{attribute 'global_init_slot' := '40510'}
VAR_GLOBAL
  LblControl_OperationMode                                     :FB_BA_Label:=( sObjName:='OPM',sDescr:='Operation Mode');
  LblControl_SummerNightCooling                                :FB_BA_Label:=( sObjName:='SNC',sDescr:='Summer night cooling');
  LblControl_DifferencePressureMonitoringSupplyAirFan          :FB_BA_Label:=( sObjName:='DPM',sDescr:='Difference Pressure Monitoring Supply Air Fan');
  LblControl_DifferencePressureMonitoringExtractAirFan         :FB_BA_Label:=( sObjName:='DPM',sDescr:='Difference Pressure Monitoring Extract Air Fan');
  LblControl_TSetpointCalculation                              :FB_BA_Label:=( sObjName:='SPC',sDescr:='Setpoint Calculation Temperature');
  LblControl_HSetpointCalculation                              :FB_BA_Label:=( sObjName:='SPC',sDescr:='Setpoint Calculation Humidity');
  LblControl_TCascadeSupplyAirControl                          :FB_BA_Label:=( sObjName:='CTL',sDescr:='Cascade control supply air temperature');
  LblControl_HCascadeSupplyAirControl                          :FB_BA_Label:=( sObjName:='CTL',sDescr:='Cascade control supply air humidity');
  LblControl_PreHeater                                         :FB_BA_Label:=( sObjName:='PRH',sDescr:='PreHeater');
  LblControl_ReHeater                                          :FB_BA_Label:=( sObjName:='RHE',sDescr:='Reheater');
  LblControl_EnergyRecovery                                    :FB_BA_Label:=( sObjName:='ERC',sDescr:='Energy Recovery');
  LblControl_SupplyAirTemperatureControl                       :FB_BA_Label:=( sObjName:='CTL',sDescr:='Supply Air Temperature Control');
  LblControl_SupplyAirDehumidifierControl                      :FB_BA_Label:=( sObjName:='CTL',sDescr:='Supply Air Dehumidification Control');
  LblControl_SupplyAirHumidifierController                     :FB_BA_Label:=( sObjName:='CTL',sDescr:='Supply Air Humidity Control');
  LblControl_SupplyAirTemperatureLimitationControl             :FB_BA_Label:=( sObjName:='CTL',sDescr:='Supply Air Temperature Limitation Control');
  LblControl_ReturnWaterControl                                :FB_BA_Label:=( sObjName:='CTL',sDescr:='Return Water Control');
  LblControl_HumidityLimitationControl                         :FB_BA_Label:=( sObjName:='CTL',sDescr:='Rel humidity limitation control');
  LblControl_CalculationPreRinseSetpoint                       :FB_BA_Label:=( sObjName:='SPC',sDescr:='Calculation PreRinse Setpoint');
  LblControl_FrostProtectionControl                            :FB_BA_Label:=( sObjName:='FPC',sDescr:='Frost Protection Control');
  LblControl_ExhaustAirTemperatureControl                      :FB_BA_Label:=( sObjName:='CTL',sDescr:='Exhaust Air Temperature Control');
  LblControl_EnergyRecoveryDeicingRamp                         :FB_BA_Label:=( sObjName:='RMP',sDescr:='Energy Recovery Deicing Ramp');
  LblControl_BACnetDevice                                      :FB_BA_Label:=( sObjName:='DEV',sDescr:='BACnet device');
  LblControl_PlantControl                                      :FB_BA_Label:=( sObjName:='PCT',sDescr:='Plant Control');
  LblControl_TSequenceControl                                  :FB_BA_Label:=( sObjName:='SEQ',sDescr:='Sequence Control Temp');
  LblControl_HSequenceControl                                  :FB_BA_Label:=( sObjName:='SEQ',sDescr:='Sequence Control Humidity');
  LblControl_GeneralBeckhoffEventClass                         :FB_BA_Label:=( sObjName:='ECL',sDescr:='Event class');
  LblControl_GeneralSettings                                   :FB_BA_Label:=( sObjName:='SYP',sDescr:='System parameters');
  LblControl_GeneralCabinetBasicEquipment                      :FB_BA_Label:=( sObjName:='CBE',sDescr:='Cabinet basic equipment');
  LblControl_GeneralCabinetAdditionalEquipment                 :FB_BA_Label:=( sObjName:='CAE',sDescr:='Cabinet additional equipment');
  LblControl_EventIndicationLamp                               :FB_BA_Label:=( sObjName:='CEM',sDescr:='Collective error message lamp');
  LblControl_AcknowledgeCommand                                :FB_BA_Label:=( sObjName:='ACK',sDescr:='Acknowledge Hardware');
  LblControl_RemoteAcknowledgement                             :FB_BA_Label:=( sObjName:='ACK',sDescr:='Remote acknowledgement fault');
  LblControl_LocalAcknowledgement                              :FB_BA_Label:=( sObjName:='ACK',sDescr:='Local acknowledgement fault');
  LblControl_Acknowledge                                       :FB_BA_Label:=( sObjName:='ACK',sDescr:='Acknowledge');
// 
  LblControl_Fuse                                              :FB_BA_Label:=( sObjName:='FUS',sDescr:='Fuse');
// Settings
  LblControl_FrostProtection                                   :FB_BA_Label:=( sObjName:='FRP',sDescr:='Frost protection');
  LblControl_MinimumOutsideTemperature                         :FB_BA_Label:=( sObjName:='TWT',sDescr:='Minimum outdoor temperature');
  LblControl_TemperatureWeatherLowLimit                        :FB_BA_Label:=( sObjName:='TWT',sDescr:='Temperature weather low limit');
  LblControl_TemperatureWeatherDamped                          :FB_BA_Label:=( sObjName:='TWD',sDescr:='Temperature weather damped');
  LblControl_TemperatureWeatherDampedLowLimit                  :FB_BA_Label:=( sObjName:='TWD',sDescr:='Temperature Weather damped low limit');
  LblControl_PressureControl                                   :FB_BA_Label:=( sObjName:='CTL',sDescr:='Pressure control');
  LblControl_Converter3Point                                   :FB_BA_Label:=( sObjName:='CNV',sDescr:='3 point converter');
  LblControl_HeatingCurve                                      :FB_BA_Label:=( sObjName:='HCV',sDescr:='Heating curve');
  LblControl_SetpointGeneration                                :FB_BA_Label:=( sObjName:='SPG',sDescr:='Setpoint generation');
  LblControl_RequestHeatState                                  :FB_BA_Label:=( sObjName:='RHS',sDescr:='Request heat state');
  LblControl_RequestHeatSetpoint                               :FB_BA_Label:=( sObjName:='RHS',sDescr:='Request heat setpoint');
  LblControl_FlowTempControl                                   :FB_BA_Label:=( sObjName:='CTL',sDescr:='Flow temperature control');
// 
  LblControl_RoomTemperatureControl                            :FB_BA_Label:=( sObjName:='RGL',sDescr:='Room Temperature Control');
  LblControl_FlowTemperatureControl                            :FB_BA_Label:=( sObjName:='CTL',sDescr:='Flow temperature control');
  LblControl_SetpointHeating                                   :FB_BA_Label:=( sObjName:='SPG',sDescr:='Setpoint generation heating');
  LblControl_SetpointCooling                                   :FB_BA_Label:=( sObjName:='SPG',sDescr:='Setpoint generation cooling');
  LblControl_Facade                                            :FB_BA_Label:=( sObjName:='FIE',sDescr:='Facade Data');
  LblControl_BuildingAlarms                                    :FB_BA_Label:=( sObjName:='FIE',sDescr:='Building Alarms');
  LblControl_BuildingEnergyLevel                               :FB_BA_Label:=( sObjName:='FIE',sDescr:='Building Energylevel');
  LblControl_BuildingMode                                      :FB_BA_Label:=( sObjName:='FIE',sDescr:='Building Operationmode');
  LblControl_BuildingSpRmT                                     :FB_BA_Label:=( sObjName:='FIE',sDescr:='Building Roomtemperature Setpoints');
  LblControl_BuildingSunprotection                             :FB_BA_Label:=( sObjName:='FIE',sDescr:='Building Sunprotection');
  LblControl_TemperatureFrost                                  :FB_BA_Label:=( sObjName:='TFR',sDescr:='Temperature Frost');
  LblControl_MixedAirStartUpRamp                               :FB_BA_Label:=( sObjName:='RMP',sDescr:='Ramp plant start');
  LblControl_Cooler                                            :FB_BA_Label:=( sObjName:='COL',sDescr:='Cooler');
  LblControl_EvtCategoryLifeSafty                              :FB_BA_Label:=( sObjName:='EDL',sDescr:='Danger to life');
  LblControl_EvtCategorySaftyMessage                           :FB_BA_Label:=( sObjName:='ESM',sDescr:='Safety message');
  LblControl_EvtCategoryAlarmMessage                           :FB_BA_Label:=( sObjName:='EAM',sDescr:='Alarm message');
  LblControl_EvtCategoryFaultMessage                           :FB_BA_Label:=( sObjName:='EFM',sDescr:='Fault message');
  LblControl_EvtCategoryMaintenanceMessage                     :FB_BA_Label:=( sObjName:='EMM',sDescr:='Maintenance message');
  LblControl_EvtCategorySystem                                 :FB_BA_Label:=( sObjName:='ESY',sDescr:='System message');
  LblControl_EvtCategoryManualOperation                        :FB_BA_Label:=( sObjName:='EMO',sDescr:='Manual operation');
  LblControl_EvtCategoryOther                                  :FB_BA_Label:=( sObjName:='EOM',sDescr:='Other message');
  LblControl_TrendLogging                                      :FB_BA_Label:=( sObjName:='TRL',sDescr:='TrendLogging                                      ');
  LblControl_WeatherParameters                                 :FB_BA_Label:=( sObjName:='WTP',sDescr:='Weather Parameters');
  LblControl_SetpointFrostProtection                           :FB_BA_Label:=( sObjName:='SP_',sDescr:='Setpoint frost protection');
  LblControl_SetpointWeatherIcing                              :FB_BA_Label:=( sObjName:='SP_',sDescr:='Setpoint icing');
  LblControl_SetpointMinimumOutsideTemperature                 :FB_BA_Label:=( sObjName:='SPI',sDescr:='Setpoint minimum outside temperature');
  LblControl_MeanDamped                                        :FB_BA_Label:=( sObjName:='MWD',sDescr:='Mean value weather temperature damped');
  LblControl_OperationalMessageTemperatureWeatherLowLimit      :FB_BA_Label:=( sObjName:='OM_',sDescr:='Operational Message Temperature Weather Low Limit');
  LblControl_OperationalMessageTemperatureWeatherDampedLowLimit:FB_BA_Label:=( sObjName:='OM_',sDescr:='Operational Message Temperature Weather Damped Low Limit');
// Beckhoff Cabinet basic equipment
  LblControl_SwitchingCommandCollectiveFaultSignalLamp         :FB_BA_Label:=( sObjName:='SC_',sDescr:='Collective fault signal lamp switching command');
  LblControl_SwitchingCommandHardwareAcknowledgement           :FB_BA_Label:=( sObjName:='SC_',sDescr:='Hardware acknowledgement switching command');
  LblControl_ButtonRemoteAcknowledgement                       :FB_BA_Label:=( sObjName:='BUT',sDescr:='Input remote acknowledgement');
  LblControl_ButtonLocalAcknowledgement                        :FB_BA_Label:=( sObjName:='BUT',sDescr:='Button acknowledgement');
// Beckhoff Heating Circuit
  LblControl_HeatingLimit                                      :FB_BA_Label:=( sObjName:='HLM',sDescr:='Heating limit ');
  LblControl_PresentOperationMode                              :FB_BA_Label:=( sObjName:='POM',sDescr:='Present operation mode');
  LblControl_OperationModeSelection                            :FB_BA_Label:=( sObjName:='OMS',sDescr:='Operation mode selection');
// Beckhoff Summer Night Cooling
  LblControl_HysteresisRoomTemperature                         :FB_BA_Label:=( sObjName:='HYS',sDescr:='Hyeresis room temperature');
  LblControl_OutsideTemperatureLowLimit                        :FB_BA_Label:=( sObjName:='MIN',sDescr:='minimum outside temperature');
  LblControl_OffValueDifferenceOutsideInsightTemperature       :FB_BA_Label:=( sObjName:='MIN',sDescr:='Off Value differenz between ouside and insight temperature');
  LblControl_OnValueDifferenceOutsideInsightTemperature        :FB_BA_Label:=( sObjName:='MAX',sDescr:='On Value differenz between ouside and insight temperature');
// Beckhoff Damper
  LblControl_DriveTimeOpen                                     :FB_BA_Label:=( sObjName:='DTO',sDescr:='Drive time open');
  LblControl_DriveTimeClose                                    :FB_BA_Label:=( sObjName:='DTC',sDescr:='Drive time close');
  LblControl_DisturbanceFeedbackOpen                           :FB_BA_Label:=( sObjName:='DSO',sDescr:='Disturbance_feedback_open');
  LblControl_DisturbanceFeedbackClose                          :FB_BA_Label:=( sObjName:='DSC',sDescr:='Disturbance_feedback_close');
// 
  LblControl_TimeDelay                                         :FB_BA_Label:=( sObjName:='TD_',sDescr:='Time delay ');
  LblControl_TimeDelayFeedback                                 :FB_BA_Label:=( sObjName:='TDF',sDescr:='Time delay feedback');
  LblControl_TimeDelayInterruptionFeedback                     :FB_BA_Label:=( sObjName:='TDI',sDescr:='Time delay interruption');
// Beckhoff pre rins
  LblControl_PreRinseDuration                                  :FB_BA_Label:=( sObjName:='PRD',sDescr:='Pre rins duration');
  LblControl_DisturbancePreRinse                               :FB_BA_Label:=( sObjName:='DST',sDescr:='Disturbance pre rinse');
  LblControl_SetpointMinimalReturnWaterTemperature             :FB_BA_Label:=( sObjName:='SP_',sDescr:='Setpoint minimal return water temperature');
// Beckhoff ramp 
  LblControl_RampTimeUp                                        :FB_BA_Label:=( sObjName:='RTU',sDescr:='Ramp time up');
  LblControl_RampTimeDown                                      :FB_BA_Label:=( sObjName:='RTD',sDescr:='Ramp time down');
  LblControl_CommandOpen                                       :FB_BA_Label:=( sObjName:='SC_',sDescr:='Switch command open');
  LblControl_CommandClose                                      :FB_BA_Label:=( sObjName:='SC_',sDescr:='Switch command close');
  LblControl_CalculatedValue                                   :FB_BA_Label:=( sObjName:='CAV',sDescr:='calculated value');
  LblControl_Value                                             :FB_BA_Label:=( sObjName:='VAL',sDescr:='Value');
// Beckhoff event class
  LblControl_EvtClass                                          :FB_BA_Label:=( sObjName:='NC_',sDescr:='Notification class');
  LblControl_FlowSwitch                                        :FB_BA_Label:=( sObjName:='OM_',sDescr:='Operating message flow monitor');
  LblControl_SmokeAlarm                                        :FB_BA_Label:=( sObjName:='DST',sDescr:='Disturbance smoke alarm');
  LblControl_SystemFailure                                     :FB_BA_Label:=( sObjName:='DST',sDescr:='Disturbance system failure');
  LblControl_Contamination                                     :FB_BA_Label:=( sObjName:='DST',sDescr:='Disturbance Contamination');
  LblControl_SwitchingCommandSmokeDetector                     :FB_BA_Label:=( sObjName:='SC_',sDescr:='Switching command acknowledge');
  LblControl_ButtonReset                                       :FB_BA_Label:=( sObjName:='BUT',sDescr:='Button acknowledge');
  LblControl_OffsetNightSetpoint                               :FB_BA_Label:=( sObjName:='ONS',sDescr:='Offset night setback');
// 
  LblControl_SetpointRelHumidityHumidification                 :FB_BA_Label:=( sObjName:='SP_',sDescr:='Setpoint Relative Humidity Humidification');
  LblControl_SetpointRelHumidityDehumidification               :FB_BA_Label:=( sObjName:='SP_',sDescr:='Setpoint Relative Humidity Dehumidification');
  LblControl_SetpointAbsHumidityHumidification                 :FB_BA_Label:=( sObjName:='SPC',sDescr:='Setpoint absolute humidity humidification');
  LblControl_SetpointAbsHumidityDehumidification               :FB_BA_Label:=( sObjName:='SPC',sDescr:='Setpoint absolute humidity dehumidification');
  LblControl_SetpointRelHumidity                               :FB_BA_Label:=( sObjName:='SP_',sDescr:='Setpoint relative humidity');
  LblControl_SetpointAbsHumidity                               :FB_BA_Label:=( sObjName:='SP_',sDescr:='Setpoint absolute humidity');
  LblControl_OperationalMessageDehumidification                :FB_BA_Label:=( sObjName:='OM_',sDescr:='Operational message dehumidification');
// 
  LblControl_SetpointSunblindPosition                          :FB_BA_Label:=( sObjName:='SP_',sDescr:='Setpoint blind position');
  LblControl_SetpointSunblindAngle                             :FB_BA_Label:=( sObjName:='SP_',sDescr:='Setpoint blind angle');
  LblControl_CommandSunblindStart                              :FB_BA_Label:=( sObjName:='SC_',sDescr:='Command sunblind start');
  LblControl_ButtonSunblind                                    :FB_BA_Label:=( sObjName:='BUT',sDescr:='Sun blind button');
  LblControl_FeedbackSunblindPosition                          :FB_BA_Label:=( sObjName:='FDB',sDescr:='Feedback blind position');
  LblControl_FeedbackSunblindAngle                             :FB_BA_Label:=( sObjName:='FDB',sDescr:='Feedback blind angle');
  LblControl_FeedbackSunblindPrio                              :FB_BA_Label:=( sObjName:='FDB',sDescr:='Feedback Telegram-Priority');
// 
  LblControl_TimeDelayStormOn                                  :FB_BA_Label:=( sObjName:='TON',sDescr:='Storm-detection time delay on');
  LblControl_TimeDelayStormOff                                 :FB_BA_Label:=( sObjName:='TOF',sDescr:='Storm-detection time delay off');
  LblControl_MaintenanceEnable                                 :FB_BA_Label:=( sObjName:='EN_',sDescr:='Maintenence positioning enable');
  LblControl_MaintenancePosition                               :FB_BA_Label:=( sObjName:='SP_',sDescr:='Setpoint maintenance position');
  LblControl_MaintenanceAngle                                  :FB_BA_Label:=( sObjName:='SP_',sDescr:='Setpoint maintenance angle');
  LblControl_FacadeThermoAutomaticEnable                       :FB_BA_Label:=( sObjName:='EN_',sDescr:='Facade-Thermoautomatic enable');
  LblControl_FacadeThermoAutomaticCoolingPosition              :FB_BA_Label:=( sObjName:='SP_',sDescr:='Facade-Thermoautomatic cooling-position');
  LblControl_FacadeThermoAutomaticCoolingAngle                 :FB_BA_Label:=( sObjName:='SP_',sDescr:='Facade-Thermoautomatic cooling-angle');
  LblControl_FacadeTwilightAutomaticEnable                     :FB_BA_Label:=( sObjName:='EN_',sDescr:='Facade-Twilightautomatic enable');
  LblControl_SunProtectionValueOn                              :FB_BA_Label:=( sObjName:='SP_',sDescr:='Sun-protection brightness on');
  LblControl_SunProtectionValueOff                             :FB_BA_Label:=( sObjName:='SP_',sDescr:='Sun-protection brightness off');
  LblControl_TimeDelaySunProtectionOn                          :FB_BA_Label:=( sObjName:='TON',sDescr:='Sun-protection brightness on');
  LblControl_TimeDelaySunProtectionOff                         :FB_BA_Label:=( sObjName:='TOF',sDescr:='Sun-protection brightness off');
  LblControl_FacadeParkingEnable                               :FB_BA_Label:=( sObjName:='EN_',sDescr:='Facade-parking enable');
  LblControl_FacadeParkingPosition                             :FB_BA_Label:=( sObjName:='SP_',sDescr:='Facade-parking position');
  LblControl_FacadeParkingAngle                                :FB_BA_Label:=( sObjName:='SP_',sDescr:='Facade-parking angle');
  LblControl_WindProtectionState                               :FB_BA_Label:=( sObjName:='STA',sDescr:='State wind-protection');
  LblControl_SunProtectionState                                :FB_BA_Label:=( sObjName:='STA',sDescr:='State sun-protection');
// 
  LblControl_LowWaterMonitor                                   :FB_BA_Label:=( sObjName:='DST',sDescr:='Low water monitor');
  LblControl_FireAlert                                         :FB_BA_Label:=( sObjName:='DST',sDescr:='Fire alert');
  LblControl_Burglary                                          :FB_BA_Label:=( sObjName:='DST',sDescr:='Burglary alert');
  LblControl_CentralSwitchOff                                  :FB_BA_Label:=( sObjName:='PLS',sDescr:='Central switch-off');
  LblControl_ForcedVentilation                                 :FB_BA_Label:=( sObjName:='PLS',sDescr:='Forced ventilation ');
  LblControl_SmokeExtraction                                   :FB_BA_Label:=( sObjName:='PLS',sDescr:='Smoke extraction');
  LblControl_SetpointIce                                       :FB_BA_Label:=( sObjName:='SP_',sDescr:='Setpoint Ice');
  LblControl_SunProtectionInterval                             :FB_BA_Label:=( sObjName:='SP_',sDescr:='Sun-protection positioning interval');
  LblControl_DeiceTime                                         :FB_BA_Label:=( sObjName:='SP_',sDescr:='Frost-protection deice-time');
  LblControl_GlobalThermoAutomaticValueOn                      :FB_BA_Label:=( sObjName:='SP_',sDescr:='Thermo-automatic radiation-value on');
  LblControl_GlobalThermoAutomaticValueOff                     :FB_BA_Label:=( sObjName:='SP_',sDescr:='Thermo-automatic radiation-value off');
  LblControl_GlobalTwilightAutomaticValueOn                    :FB_BA_Label:=( sObjName:='SP_',sDescr:='Twilight-automatic brightness-value on');
  LblControl_GlobalTwilightAutomaticValueOff                   :FB_BA_Label:=( sObjName:='SP_',sDescr:='Twilight-automatic brightness-value on');
  LblControl_IceAlert                                          :FB_BA_Label:=( sObjName:='DST',sDescr:='Ice alert');
  LblControl_GlobalThermoAutomaticRelease                      :FB_BA_Label:=( sObjName:='EN_',sDescr:='Thermo-automatic release');
  LblControl_GlobalTwilightAutomaticRelease                    :FB_BA_Label:=( sObjName:='EN_',sDescr:='Twilight-automatic release');
  LblControl_GlobalResetManMode                                :FB_BA_Label:=( sObjName:='PLS',sDescr:='Global Reset Manual Mode');
// 
  LblControl_BuildingEnergyLevelManual                         :FB_BA_Label:=( sObjName:='OPS',sDescr:='Building-energy-level manual selection');
  LblControl_BuildingEnergyLevelActual                         :FB_BA_Label:=( sObjName:='POM',sDescr:='Building-energy-level actual selection');
  LblControl_BuildingEnergyLevelSched                          :FB_BA_Label:=( sObjName:='SCH',sDescr:='Building-energy-level scheduler');
  LblControl_BuildingModeManual                                :FB_BA_Label:=( sObjName:='OPS',sDescr:='Building-mode manual selection');
  LblControl_BuildingModeActual                                :FB_BA_Label:=( sObjName:='POM',sDescr:='Building-mode actual selection');
  LblControl_BuildingModeSched                                 :FB_BA_Label:=( sObjName:='SCH',sDescr:='Building-mode scheduler');
// 
  LblControl_SummerCompensationX1                              :FB_BA_Label:=( sObjName:='IPX',sDescr:='Summercompensation X1');
  LblControl_SummerCompensationX2                              :FB_BA_Label:=( sObjName:='IPX',sDescr:='Summercompensation X2');
  LblControl_SummerCompensationY1                              :FB_BA_Label:=( sObjName:='IPY',sDescr:='Summercompensation Y1');
  LblControl_SummerCompensationY2                              :FB_BA_Label:=( sObjName:='IPY',sDescr:='Summercompensation Y2');
  LblControl_WinterCompensationX1                              :FB_BA_Label:=( sObjName:='IPX',sDescr:='Wintercompensation X1');
  LblControl_WinterCompensationX2                              :FB_BA_Label:=( sObjName:='IPX',sDescr:='Wintercompensation X2');
  LblControl_WinterCompensationY1                              :FB_BA_Label:=( sObjName:='IPY',sDescr:='Wintercompensation Y1');
  LblControl_WinterCompensationY2                              :FB_BA_Label:=( sObjName:='IPY',sDescr:='Wintercompensation Y2');
  LblControl_SummerCompensation                                :FB_BA_Label:=( sObjName:='SCP',sDescr:='SummerCompensation');
  LblControl_WinterCompensation                                :FB_BA_Label:=( sObjName:='WCP',sDescr:='WinterCompensation');
  LblControl_SummerCompensationYmin                            :FB_BA_Label:=( sObjName:='SPI',sDescr:='Summer Compensation Ymin');
  LblControl_SummerCompensationYmax                            :FB_BA_Label:=( sObjName:='SPX',sDescr:='Summer Compensation Ymax');
  LblControl_WinterCompensationYmin                            :FB_BA_Label:=( sObjName:='SPI',sDescr:='Winter Compensation Ymin');
  LblControl_WinterCompensationYmax                            :FB_BA_Label:=( sObjName:='SPX',sDescr:='Winter Compensation Ymax');
  LblControl_SummerCompensationSp                              :FB_BA_Label:=( sObjName:='SPC',sDescr:='Summer Compensation Setpoint');
  LblControl_WinterCompensationSp                              :FB_BA_Label:=( sObjName:='SPC',sDescr:='Winter Compensation Setpoint');
  LblControl_SetpointShiftHeating                              :FB_BA_Label:=( sObjName:='SP_',sDescr:='Setpoint shift heating');
  LblControl_SetpointShiftCooling                              :FB_BA_Label:=( sObjName:='SP_',sDescr:='Setpoint shift cooling');
  LblControl_DampConstant                                      :FB_BA_Label:=( sObjName:='SP_',sDescr:='Damp constant');
// 
  LblControl_DelayOn                                           :FB_BA_Label:=( sObjName:='TON',sDescr:='Switch-on delay');
  LblControl_DelayOff                                          :FB_BA_Label:=( sObjName:='TOF',sDescr:='Switch-off delay');
  LblControl_AntiBlocking                                      :FB_BA_Label:=( sObjName:='ABK',sDescr:='Anti Blocking');
  LblControl_IdlePeriod                                        :FB_BA_Label:=( sObjName:='ITV',sDescr:='Idle Period');
  LblControl_ImpulsLength                                      :FB_BA_Label:=( sObjName:='IPL',sDescr:='Impuls length');
  LblControl_SuppyAirTempSetpointHeaterCalc                    :FB_BA_Label:=( sObjName:='SPC',sDescr:='Suppy Air Sp Heater Calc');
  LblControl_SuppyAirTempSetpointCoolerCalc                    :FB_BA_Label:=( sObjName:='SPC',sDescr:='Suppy Air Sp Cooler Calc');
  LblControl_SuppyAirTempSetpointERCCalc                       :FB_BA_Label:=( sObjName:='SPC',sDescr:='Suppy Air Sp ERC Calc');
  LblControl_X01                                               :FB_BA_Label:=( sObjName:='SPX',sDescr:='Value Base [X1]');
  LblControl_X02                                               :FB_BA_Label:=( sObjName:='SPX',sDescr:='Value Base [X2]');
  LblControl_X03                                               :FB_BA_Label:=( sObjName:='SPX',sDescr:='Value Base [X3]');
  LblControl_X04                                               :FB_BA_Label:=( sObjName:='SPX',sDescr:='Value Base [X4]');
  LblControl_X05                                               :FB_BA_Label:=( sObjName:='SPX',sDescr:='Value Base [X5]');
  LblControl_X06                                               :FB_BA_Label:=( sObjName:='SPX',sDescr:='Value Base [X6]');
  LblControl_X07                                               :FB_BA_Label:=( sObjName:='SPX',sDescr:='Value Base [X7]');
  LblControl_Y01                                               :FB_BA_Label:=( sObjName:='SPY',sDescr:='Value Base [Y1]');
  LblControl_Y02                                               :FB_BA_Label:=( sObjName:='SPY',sDescr:='Value Base [Y2]');
  LblControl_Y02_03                                            :FB_BA_Label:=( sObjName:='SPY',sDescr:='Value Base [Y2Y3]');
  LblControl_Y03                                               :FB_BA_Label:=( sObjName:='SPY',sDescr:='Value Base [Y3]');
  LblControl_Y04                                               :FB_BA_Label:=( sObjName:='SPY',sDescr:='Value Base [Y4]');
  LblControl_Y05                                               :FB_BA_Label:=( sObjName:='SPY',sDescr:='Value Base [Y5]');
  LblControl_Y06                                               :FB_BA_Label:=( sObjName:='SPY',sDescr:='Value Base [Y6]');
  LblControl_Y07                                               :FB_BA_Label:=( sObjName:='SPY',sDescr:='Value Base [Y7]');
  LblControl_FeedbackMonitoring                                :FB_BA_Label:=( sObjName:='FDM',sDescr:='Feedback monitoring');
  LblControl_PreAlarmLimitMAX                                  :FB_BA_Label:=( sObjName:='LMX',sDescr:='Pre Alarm Limit MAX');
  LblControl_PreAlarmLimitMIN                                  :FB_BA_Label:=( sObjName:='LMI',sDescr:='Pre Alarm Limit MIN');
  LblControl_PreAlarmFault                                     :FB_BA_Label:=( sObjName:='DST',sDescr:='Pre Alarm Fault');
  LblControl_MainAlarmLimitMAX                                 :FB_BA_Label:=( sObjName:='LMX',sDescr:='Main Alarm Limit MAX');
  LblControl_MainAlarmLimitMIN                                 :FB_BA_Label:=( sObjName:='LMI',sDescr:='Main Alarm Limit MIN');
  LblControl_MainAlarmFault                                    :FB_BA_Label:=( sObjName:='DST',sDescr:='Main Alarm Fault');
  LblControl_ProcPreRinse                                      :FB_BA_LabelProcess:=( sProcessName:='Process Pre Rinse');
  LblControl_ProjectInfo                                       :FB_BA_Label:=( sObjName:='PI_',sDescr:='Project Info');
END_VAR

// ---- Templates/GVLs/Language/English/LblFunctions_EN.TcGVL
{region '#Template'}
	{attribute 'Version' := '1.2.0.0'}
	{attribute 'Tags' := '"LCID": "1031", "Text": "GVL, AKS, Labels, ObjectName, Description"'}
	{attribute 'Tags' := '"LCID": "1033", "Text": "GVL, DPAD, Labels, ObjectName, Description"'}
	{attribute 'Description' := '"LCID": "1031", "Text": "Anlagenkennzeichnungssystem, Labels functions"'}
	{attribute 'Description' := '"LCID": "1033", "Text": "Data Point Addressing Description, Labels functions"'}
{endregion}

{attribute 'global_init_slot' := '40510'}
VAR_GLOBAL
  LblFunctions_Requirement                                       :FB_BA_Label:=( sObjName:='REQ',sDescr:='Requirement');
  LblFunctions_SystemSwitch                                      :FB_BA_Label:=( sObjName:='PLS',sDescr:='Plant switch');
  LblFunctions_StatusOccupiedRoom                                :FB_BA_Label:=( sObjName:='OCC',sDescr:='Occupied status room');
  LblFunctions_LimitCalculatedValue                              :FB_BA_Label:=( sObjName:='LMC',sDescr:='Calculated limit value');
  LblFunctions_SetpointCalculated                                :FB_BA_Label:=( sObjName:='SPC',sDescr:='Calculated setpoint');
  LblFunctions_ReadyForOperation                                 :FB_BA_Label:=( sObjName:='RFO',sDescr:='Ready for operation');
  LblFunctions_OperationalMessage                                :FB_BA_Label:=( sObjName:='OM_',sDescr:='Operational message');
  LblFunctions_HoursOfOperation                                  :FB_BA_Label:=( sObjName:='OH_',sDescr:='Operating hours');
  LblFunctions_LimitValueHoursOfOperation                        :FB_BA_Label:=( sObjName:='OHL',sDescr:='Operating hours limit value');
  LblFunctions_ObjectCalendar                                    :FB_BA_Label:=( sObjName:='CAL',sDescr:='Calendar object');
  LblFunctions_ObjectCommand                                     :FB_BA_Label:=( sObjName:='COM',sDescr:='Command object');
  LblFunctions_DifferentialConstantController                    :FB_BA_Label:=( sObjName:='TV_',sDescr:='Differential constant controller');
  LblFunctions_SwitchOnErrorUnauthorisedON                       :FB_BA_Label:=( sObjName:='SWE',sDescr:='Switch-on error, unauthorised ON');
  LblFunctions_EnergyLevel                                       :FB_BA_Label:=( sObjName:='EL_',sDescr:='Energy level');
  LblFunctions_EnergyLevelCalculated                             :FB_BA_Label:=( sObjName:='ELC',sDescr:='Energy level calculated');
  LblFunctions_UnlockingDevice                                   :FB_BA_Label:=( sObjName:='UNL',sDescr:='Unlocking device');
  LblFunctions_ObjectEventEnrollment                             :FB_BA_Label:=( sObjName:='EE_',sDescr:='Event enrollment object');
  LblFunctions_Enabled                                           :FB_BA_Label:=( sObjName:='EN_',sDescr:='Enabled');
  LblFunctions_DangerAlarm                                       :FB_BA_Label:=( sObjName:='DA_',sDescr:='Danger alarm');
  LblFunctions_Threshold                                         :FB_BA_Label:=( sObjName:='LM_',sDescr:='Limit value');
  LblFunctions_LimitMAX                                          :FB_BA_Label:=( sObjName:='LMX',sDescr:='MAX limit');
  LblFunctions_LimitMIN                                          :FB_BA_Label:=( sObjName:='LMI',sDescr:='MIN limit');
  LblFunctions_LimitNight                                        :FB_BA_Label:=( sObjName:='LMN',sDescr:='Night limit');
  LblFunctions_LimitDay                                          :FB_BA_Label:=( sObjName:='LMD',sDescr:='Day limit');
  LblFunctions_ObjectGroup                                       :FB_BA_Label:=( sObjName:='GP_',sDescr:='Group object');
  LblFunctions_localPriorityAndOperatingUnitsManualMessage       :FB_BA_Label:=( sObjName:='MNM',sDescr:='local priority and operating units manual message');
  LblFunctions_HeatingCharacteristicCurveExponent                :FB_BA_Label:=( sObjName:='HEX',sDescr:='Heating characteristic curve exponent');
  LblFunctions_HeatingCharacteristicCurveParallelDisplacement    :FB_BA_Label:=( sObjName:='HPD',sDescr:='Heating characteristic curve parallel displacement');
  LblFunctions_HeatingCharacteristicCurveSteepness               :FB_BA_Label:=( sObjName:='HST',sDescr:='Heating characteristic curve steepness');
  LblFunctions_HeatingCircuitNightReduction                      :FB_BA_Label:=( sObjName:='NGT',sDescr:='Heating circuit night reduction');
  LblFunctions_Hysteresis                                        :FB_BA_Label:=( sObjName:='HYS',sDescr:='Hysteresis');
  LblFunctions_Calendar                                          :FB_BA_Label:=( sObjName:='CAL',sDescr:='Calendar');
  LblFunctions_RuntimeError                                      :FB_BA_Label:=( sObjName:='RUN',sDescr:='Runtime error');
  LblFunctions_LoopMAXLimit                                      :FB_BA_Label:=( sObjName:='LPX',sDescr:='Loop MAX limit');
  LblFunctions_LoopMINLimit                                      :FB_BA_Label:=( sObjName:='LPI',sDescr:='Loop MIN limit');
  LblFunctions_LoopObject                                        :FB_BA_Label:=( sObjName:='LP_',sDescr:='Loop object (controller object) – complex object');
  LblFunctions_LoopObjectCascadeSupplyAirTemperature             :FB_BA_Label:=( sObjName:='LP_',sDescr:='Cascade controller supply air temperature ');
  LblFunctions_LoopObjectCascadeSupplyAirHumidity                :FB_BA_Label:=( sObjName:='LP_',sDescr:='Cascade controller supply air humidity ');
  LblFunctions_MaximumValue                                      :FB_BA_Label:=( sObjName:='MAX',sDescr:='Maximum value');
  LblFunctions_MeasuredValue                                     :FB_BA_Label:=( sObjName:='MV_',sDescr:='Measured value');
  LblFunctions_MeasuredValueCalculated                           :FB_BA_Label:=( sObjName:='MVC',sDescr:='Measured value calculated');
  LblFunctions_MeasuredValueEast                                 :FB_BA_Label:=( sObjName:='MV_',sDescr:='Measured value East');
  LblFunctions_MeasuredValueNorth                                :FB_BA_Label:=( sObjName:='MV_',sDescr:='Measured value North');
  LblFunctions_MeasuredValueSouth                                :FB_BA_Label:=( sObjName:='MV_',sDescr:='Measured value South');
  LblFunctions_MeasuredValueWest                                 :FB_BA_Label:=( sObjName:='MV_',sDescr:='Measured value West');
  LblFunctions_MinimumValue                                      :FB_BA_Label:=( sObjName:='MIN',sDescr:='Minimum value');
  LblFunctions_Mean                                              :FB_BA_Label:=( sObjName:='MVL',sDescr:='Mean value');
  LblFunctions_FollowUpTime                                      :FB_BA_Label:=( sObjName:='FUT',sDescr:='Follow-up time');
  LblFunctions_ResetTime                                         :FB_BA_Label:=( sObjName:='RST',sDescr:='Reset time');
  LblFunctions_FeedbackDelay                                     :FB_BA_Label:=( sObjName:='TDF',sDescr:='Time delay feedback');
  LblFunctions_ObjectNotificationClass                           :FB_BA_Label:=( sObjName:='NC_',sDescr:='Notification class object');
  LblFunctions_EventClassObject                                  :FB_BA_Label:=( sObjName:='ECL',sDescr:='Event class');
  LblFunctions_Programobject                                     :FB_BA_Label:=( sObjName:='PRG',sDescr:='Program');
  LblFunctions_ProportionalBand                                  :FB_BA_Label:=( sObjName:='XP_',sDescr:='Proportional band');
  LblFunctions_FeedbackOPEN                                      :FB_BA_Label:=( sObjName:='FDO',sDescr:='Feedback OPEN');
  LblFunctions_FeedbackCLOSED                                    :FB_BA_Label:=( sObjName:='FDC',sDescr:='Feedback CLOSED');
  LblFunctions_FeedbackValue                                     :FB_BA_Label:=( sObjName:='FDB',sDescr:='Feedback value');
  LblFunctions_FeedbackErrorOPEN                                 :FB_BA_Label:=( sObjName:='FEO',sDescr:='Feedback error OPEN');
  LblFunctions_FeedbackErrorCLOSED                               :FB_BA_Label:=( sObjName:='FEC',sDescr:='Feedback error CLOSED');
  LblFunctions_Feedback                                          :FB_BA_Label:=( sObjName:='FDB',sDescr:='Feedback');
  LblFunctions_ExecutionControl                                  :FB_BA_Label:=( sObjName:='EXC',sDescr:='Execution control');
  LblFunctions_SwitchingCommand                                  :FB_BA_Label:=( sObjName:='SC_',sDescr:='Switching command');
  LblFunctions_Scheduler                                         :FB_BA_Label:=( sObjName:='SCH',sDescr:='Scheduler');
  LblFunctions_Setpoint                                          :FB_BA_Label:=( sObjName:='SP_',sDescr:='Setpoint');
  LblFunctions_SetpointComfortHeating                            :FB_BA_Label:=( sObjName:='SP_',sDescr:='Setpoint comfort heating');
  LblFunctions_SetpointPreComfortHeating                         :FB_BA_Label:=( sObjName:='SP_',sDescr:='Setpoint pre-comfort heating');
  LblFunctions_SetpointEconomyHeating                            :FB_BA_Label:=( sObjName:='SP_',sDescr:='Setpoint economy heating');
  LblFunctions_SetpointProtectionHeating                         :FB_BA_Label:=( sObjName:='SP_',sDescr:='Setpoint protection heating');
  LblFunctions_SetpointComfortCooling                            :FB_BA_Label:=( sObjName:='SP_',sDescr:='Setpoint comfort cooling');
  LblFunctions_SetpointPreComfortCooling                         :FB_BA_Label:=( sObjName:='SP_',sDescr:='Setpoint pre-comfort cooling');
  LblFunctions_SetpointEconomyCooling                            :FB_BA_Label:=( sObjName:='SP_',sDescr:='Setpoint economy cooling');
  LblFunctions_SetpointProtectionCooling                         :FB_BA_Label:=( sObjName:='SP_',sDescr:='Setpoint protection cooling');
  LblFunctions_SetpointBase                                      :FB_BA_Label:=( sObjName:='SPB',sDescr:='Base setpoint');
  LblFunctions_SetpointHeating                                   :FB_BA_Label:=( sObjName:='SPH',sDescr:='Heating setpoint');
  LblFunctions_SetpointCooling                                   :FB_BA_Label:=( sObjName:='SPC',sDescr:='Cooling setpoint');
  LblFunctions_SetpointMaximum                                   :FB_BA_Label:=( sObjName:='SPX',sDescr:='Setpoint, maximum');
  LblFunctions_SetpointMechanical                                :FB_BA_Label:=( sObjName:='SPM',sDescr:='Setpoint, mechanical');
  LblFunctions_SetpointMinimum                                   :FB_BA_Label:=( sObjName:='SPI',sDescr:='Setpoint, minimum');
  LblFunctions_SetpointNight                                     :FB_BA_Label:=( sObjName:='SPN',sDescr:='Night setpoint');
  LblFunctions_SetpointDay                                       :FB_BA_Label:=( sObjName:='SPD',sDescr:='Day setpoint');
  LblFunctions_SetpointAdjuster                                  :FB_BA_Label:=( sObjName:='SPA',sDescr:='Setpoint adjuster');
  LblFunctions_SetpointAdjustmentMechanical                      :FB_BA_Label:=( sObjName:='SPA',sDescr:='Setpoint adjustment, mechanical');
  LblFunctions_Selection                                         :FB_BA_Label:=( sObjName:='SEL',sDescr:='Selection');
  LblFunctions_Status                                            :FB_BA_Label:=( sObjName:='STA',sDescr:='Status');
  LblFunctions_ControlSignal                                     :FB_BA_Label:=( sObjName:='CS_',sDescr:='Control signal');
  LblFunctions_Fault                                             :FB_BA_Label:=( sObjName:='FAU',sDescr:='Fault');
  LblFunctions_FaultFuse                                         :FB_BA_Label:=( sObjName:='FAU',sDescr:='Fuse fault ');
  LblFunctions_Button                                            :FB_BA_Label:=( sObjName:='BUT',sDescr:='Button');
  LblFunctions_DeadZone                                          :FB_BA_Label:=( sObjName:='DZ_',sDescr:='Dead zone');
  LblFunctions_ObjectTrendLogMultiple                            :FB_BA_Label:=( sObjName:='TRM',sDescr:='Trend log multiple object');
  LblFunctions_ObjectTrendLog                                    :FB_BA_Label:=( sObjName:='TR_',sDescr:='Trend log object');
  LblFunctions_AmplificationController                           :FB_BA_Label:=( sObjName:='KP_',sDescr:='Amplification controller');
  LblFunctions_RetentionPeriod                                   :FB_BA_Label:=( sObjName:='TV_',sDescr:='Retention period');
  LblFunctions_MaintenanceMessage                                :FB_BA_Label:=( sObjName:='MTM',sDescr:='Maintenance message');
  LblFunctions_Efficiency                                        :FB_BA_Label:=( sObjName:='EFC',sDescr:='Efficiency');
  LblFunctions_CountValue                                        :FB_BA_Label:=( sObjName:='CNT',sDescr:='Count value');
  LblFunctions_TimeProgram                                       :FB_BA_Label:=( sObjName:='TPR',sDescr:='Time program');
// Beckhoff Scale
  LblFunctions_ValueX1                                           :FB_BA_Label:=( sObjName:='IPX',sDescr:='Value interpolation point [X1]');
  LblFunctions_ValueX2                                           :FB_BA_Label:=( sObjName:='IPX',sDescr:='Value interpolation point [X2]');
  LblFunctions_ValueX3                                           :FB_BA_Label:=( sObjName:='IPX',sDescr:='Value interpolation point [X3]');
  LblFunctions_ValueX4                                           :FB_BA_Label:=( sObjName:='IPX',sDescr:='Value interpolation point [X4]');
  LblFunctions_ValueX5                                           :FB_BA_Label:=( sObjName:='IPX',sDescr:='Value interpolation point [X4]');
  LblFunctions_ValueX6                                           :FB_BA_Label:=( sObjName:='IPX',sDescr:='Value interpolation point [X4]');
  LblFunctions_ValueX7                                           :FB_BA_Label:=( sObjName:='IPX',sDescr:='Value interpolation point [X4]');
  LblFunctions_ValueY1                                           :FB_BA_Label:=( sObjName:='IPY',sDescr:='Value interpolation point [Y1]');
  LblFunctions_ValueY2                                           :FB_BA_Label:=( sObjName:='IPY',sDescr:='Value interpolation point [Y2]');
  LblFunctions_ValueY3                                           :FB_BA_Label:=( sObjName:='IPY',sDescr:='Value interpolation point [Y3]');
  LblFunctions_ValueY2_3                                         :FB_BA_Label:=( sObjName:='IPY',sDescr:='Value interpolation point [Y2-Y3]');
  LblFunctions_ValueY4                                           :FB_BA_Label:=( sObjName:='IPY',sDescr:='Value interpolation point [Y4]');
  LblFunctions_ValueY5                                           :FB_BA_Label:=( sObjName:='IPY',sDescr:='Value interpolation point [Y4]');
  LblFunctions_ValueY6                                           :FB_BA_Label:=( sObjName:='IPY',sDescr:='Value interpolation point [Y4]');
  LblFunctions_ValueY7                                           :FB_BA_Label:=( sObjName:='IPY',sDescr:='Value interpolation point [Y4]');
  LblFunctions_SuppyAirTempSetpointHeaterCalc                    :FB_BA_Label:=( sObjName:='SPC',sDescr:='Supply air Temperature setpoint heater calculated');
  LblFunctions_SuppyAirTempSetpointCoolerCalc                    :FB_BA_Label:=( sObjName:='SPC',sDescr:='Supply air Temperature setpoint cooler calculated');
  LblFunctions_SuppyAirTempSetpointERCCalc                       :FB_BA_Label:=( sObjName:='SPC',sDescr:='Supply air Temperature setpoint ERC calculated');
END_VAR

// ---- Templates/GVLs/Language/English/TxtEvent_EN.TcGVL
{region '#Template'}
	{attribute 'Version' := '1.2.0.0'}
	{attribute 'Tags' := '"LCID": "1031", "Text": "GVL, Property, Event, Event Message Text, Active Text, Inactive Text"'}
	{attribute 'Tags' := '"LCID": "1033", "Text": "GVL, Property, Event, Event Message Text, Active Text, Inactive Text"'}
	{attribute 'Description' := '"LCID": "1031", "Text": "Textliste Properties Event Message Text, Active Text, Inactive Text"'}
	{attribute 'Description' := '"LCID": "1033", "Text": "Text list Properties Event Message Text, Active Text, Inactive Text"'}
{endregion}

{attribute 'global_init_slot' := '40510'}
VAR_GLOBAL
  txtEvent_No                                                :T_BA_StateText:='No';
  txtEvent_Yes                                               :T_BA_StateText:='Yes';
  txtEvent_Auto                                              :T_BA_StateText:='Auto';
  txtEvent_Manual                                            :T_BA_StateText:='Manual';
  txtEvent_Off                                               :T_BA_StateText:='Off';
  txtEvent_On                                                :T_BA_StateText:='On';
  txtEvent_Opened                                            :T_BA_StateText:='Opened';
  txtEvent_Closed                                            :T_BA_StateText:='Closed';
  txtEvent_Open                                              :T_BA_StateText:='Open';
  txtEvent_Close                                             :T_BA_StateText:='Close';
  txtEvent_Step1                                             :T_BA_StateText:='Step1';
  txtEvent_Step2                                             :T_BA_StateText:='Step2';
  txtEvent_Step3                                             :T_BA_StateText:='Step3';
  txtEvent_Step4                                             :T_BA_StateText:='Step4';
  txtEvent_Step5                                             :T_BA_StateText:='Step5';
  txtEvent_Step6                                             :T_BA_StateText:='Step6';
  txtEvent_Step7                                             :T_BA_StateText:='Step7';
  txtEvent_Step8                                             :T_BA_StateText:='Step8';
  txtEvent_Released                                          :T_BA_StateText:='Released';
  txtEvent_Inactive                                          :T_BA_StateText:='Inactive';
  txtEvent_Active                                            :T_BA_StateText:='Active';
  txtEvent_Normal                                            :T_BA_StateText:='Normal';
  txtEvent_Offnormal                                         :T_BA_StateText:='Offnormal';
  txtEvent_Alert                                             :T_BA_StateText:='Alert';
  txtEvent_Disturb                                           :T_BA_StateText:='Disturb';
  txtEvent_Error                                             :T_BA_StateText:='Error';
  txtEvent_Triggered                                         :T_BA_StateText:='Triggered';
  txtEvent_Maintenace                                        :T_BA_StateText:='Maintenace';
  txtEvent_Exceeded                                          :T_BA_StateText:='Exceeded';
  txtEvent_Monitoring                                        :T_BA_StateText:='Monitoring';
  txtEvent_Protection                                        :T_BA_StateText:='Protection';
  txtEvent_Economy                                           :T_BA_StateText:='Economy';
  txtEvent_PreComfort                                        :T_BA_StateText:='PreComfort';
  txtEvent_Comfort                                           :T_BA_StateText:='Comfort';
  txtEvent_Reached                                           :T_BA_StateText:='Reached';
  txtEvent_NotReached                                        :T_BA_StateText:='NotReached';
  txtEvent_None                                              :T_BA_StateText:='None';
  txtEvent_EmergencyStop                                     :T_BA_StateText:='EmergencyStop';
  txtEvent_Frost                                             :T_BA_StateText:='Frost';
  txtEvent_SmokeExtraction_P                                 :T_BA_StateText:='SmokeExtraction_P';
  txtEvent_SmokeExtractionSupplyAir                          :T_BA_StateText:='SmokeExtractionSupplyAir';
  txtEvent_SmokeExtractionExtractAir                         :T_BA_StateText:='SmokeExtractionExtractAir';
  txtEvent_CoolDownProtection                                :T_BA_StateText:='CoolDownProtection';
  txtEvent_OverHeatingProtection                             :T_BA_StateText:='OverHeatingProtection';
  txtEvent_Fire                                              :T_BA_StateText:='Fire';
  txtEvent_NightCooling                                      :T_BA_StateText:='NightCooling';
  txtEvent_ForcedVentilation                                 :T_BA_StateText:='ForcedVentilation';
  txtEvent_CentralSwitchOff                                  :T_BA_StateText:='CentralSwitchOff';
  txtEvent_Locked                                            :T_BA_StateText:='Locked';
  txtEvent_Contaminated                                      :T_BA_StateText:='Contaminated';
  txtEvent_Stop                                              :T_BA_StateText:='Stop';
  txtEvent_Critical                                          :T_BA_StateText:='Critical';
  txtEvent_UnCiritical                                       :T_BA_StateText:='UnCiritical';
  txtEvent_Average                                           :T_BA_StateText:='Average';
  txtEvent_HeatCool                                          :T_BA_StateText:='HeatCool';
  txtEvent_AverageHeatCool                                   :T_BA_StateText:='AverageHeatCool';
  txtEvent_Direction                                         :T_BA_StateText:='Direction';
  txtEvent_Default                                           :T_BA_StateText:='Default';
  txtEvent_Cleaning                                          :T_BA_StateText:='Cleaning';
  txtEvent_Nightwatch                                        :T_BA_StateText:='Nightwatch';
  txtEvent_SupplyAirTControlReheater                         :T_BA_StateText:='Supply air temp control reheater';
  txtEvent_SupplyAirTControlPreheater                        :T_BA_StateText:='Supply air temp control preheater';
  txtEvent_SupplyAirTControlERC                              :T_BA_StateText:='Supply air temp control ERC';
  txtEvent_SupplyAirTControlMix                              :T_BA_StateText:='Supply air temp control mixed air';
  txtEvent_SupplyAirTControlCooler                           :T_BA_StateText:='Supply air temp control cooler';
  txtEvent_SupplyAirXControlCooler                           :T_BA_StateText:='Supply air humidity control cooler';
  txtEvent_SupplyAirXControlHumf                             :T_BA_StateText:='Supply air humidity control humidifier';
END_VAR

// ---- Templates/GVLs/Language/English/TxtPlant_EN.TcGVL
{region '#Template'}
	{attribute 'Version' := '1.2.0.0'}
	{attribute 'Tags' := '"LCID": "1031", "Text": "GVL, DPAD, Plants, ObjectName, Description"'}
	{attribute 'Tags' := '"LCID": "1033", "Text": "GVL, DPAD, Plants, ObjectName, Description"'}
	{attribute 'Description' := '"LCID": "1031", "Text": "Textliste Anlagen"'}
	{attribute 'Description' := '"LCID": "1033", "Text": "Text list plants"'}
{endregion}

{attribute 'global_init_slot' := '40510'}
VAR_GLOBAL
  TxTPlant_Facade_sObjectName                                            :T_BA_StateText:='FAC';
  TxTPlant_Facade_sDescription                                            :T_BA_StateText:='Facade';
  TxTPlant_Natural_smoke_extraction_sObjectName                          :T_BA_StateText:='NSE';
  TxTPlant_Natural_smoke_extraction_sDescription                          :T_BA_StateText:='Natural smoke extraction';
  TxTPlant_Doors_gates_sluices_sObjectName                               :T_BA_StateText:='DGS';
  TxTPlant_Doors_gates_sluices_sDescription                               :T_BA_StateText:='Doors, gates, sluices';
  TxTPlant_Smoke_and_heat_extraction_system_sObjectName                  :T_BA_StateText:='SHV';
  TxTPlant_Smoke_and_heat_extraction_system_sDescription                  :T_BA_StateText:='Smoke and heat extraction system';
  TxTPlant_Sunlight_protection_sObjectName                               :T_BA_StateText:='SUN';
  TxTPlant_Sunlight_protection_sDescription                               :T_BA_StateText:='Sunlight protection';
// 411 Sewage plants
  TxTPlant_Separator_facility_sObjectName                                :T_BA_StateText:='SEP';
  TxTPlant_Separator_facility_sDescription                                :T_BA_StateText:='Separator facility';
  TxTPlant_Lifting_system_sObjectName                                    :T_BA_StateText:='LIF';
  TxTPlant_Lifting_system_sDescription                                    :T_BA_StateText:='Lifting system';
  TxTPlant_Neutralisation_plant_sObjectName                              :T_BA_StateText:='NEU';
  TxTPlant_Neutralisation_plant_sDescription                              :T_BA_StateText:='Neutralisation plant';
// 412 water plants
  TxTPlant_Trace_heating_sObjectName                                     :T_BA_StateText:='TRH';
  TxTPlant_Trace_heating_sDescription                                     :T_BA_StateText:='Trace heating';
  TxTPlant_Process_water_sObjectName                                     :T_BA_StateText:='PCW';
  TxTPlant_Process_water_sDescription                                     :T_BA_StateText:='Process water';
  TxTPlant_Well_water_sObjectName                                        :T_BA_StateText:='WWT';
  TxTPlant_Well_water_sDescription                                        :T_BA_StateText:='Well water';
  TxTPlant_Dispensing_installation_sObjectName                           :T_BA_StateText:='DPS';
  TxTPlant_Dispensing_installation_sDescription                           :T_BA_StateText:='Dispensing installation';
  TxTPlant_Pressure_booster_system_sObjectName                           :T_BA_StateText:='PBS';
  TxTPlant_Pressure_booster_system_sDescription                           :T_BA_StateText:='Pressure booster system';
  TxTPlant_Softening_unit_sObjectName                                    :T_BA_StateText:='SOU';
  TxTPlant_Softening_unit_sDescription                                    :T_BA_StateText:='Softening unit';
// Drinking water
  TxTPlant_Drinking_water_heating_system_sObjectName                     :T_BA_StateText:='DWH';
  TxTPlant_Drinking_water_heating_system_sDescription                     :T_BA_StateText:='Drinking water heating system';
  TxTPlant_Reverse_osmosis_system_sObjectName                            :T_BA_StateText:='ROS';
  TxTPlant_Reverse_osmosis_system_sDescription                            :T_BA_StateText:='Reverse osmosis system';
  TxTPlant_Desalination_plant_sObjectName                                :T_BA_StateText:='SAP';
  TxTPlant_Desalination_plant_sDescription                                :T_BA_StateText:='Desalination plant';
// 421 Heat generation plants
  TxTPlant_BHKW_sObjectName                                              :T_BA_StateText:='BHK';
  TxTPlant_BHKW_sDescription                                              :T_BA_StateText:='BHKW';
  TxTPlant_Electric_heating_sObjectName                                  :T_BA_StateText:='EHT';
  TxTPlant_Electric_heating_sDescription                                  :T_BA_StateText:='Electric heating';
  TxTPlant_District_heating_transfer_sObjectName                         :T_BA_StateText:='DHT';
  TxTPlant_District_heating_transfer_sDescription                         :T_BA_StateText:='District heating transfer';
// Geothermal system
  TxTPlant_Boiler_sObjectName                                            :T_BA_StateText:='BOI';
  TxTPlant_Boiler_sDescription                                            :T_BA_StateText:='Boiler';
  TxTPlant_Clean_steam_generation_sObjectName                            :T_BA_StateText:='CSG';
  TxTPlant_Clean_steam_generation_sDescription                            :T_BA_StateText:='Clean steam generation';
  TxTPlant_Solar_power_system_sObjectName                                :T_BA_StateText:='SOL';
  TxTPlant_Solar_power_system_sDescription                                :T_BA_StateText:='Solar power system';
  TxTPlant_Heating_pump_sObjectName                                      :T_BA_StateText:='HPU';
  TxTPlant_Heating_pump_sDescription                                      :T_BA_StateText:='Heating pump';
// 422 Heat distribution networks
  TxTPlant_Pressure_maintenance_sObjectName                              :T_BA_StateText:='PMT';
  TxTPlant_Pressure_maintenance_sDescription                              :T_BA_StateText:='Pressure maintenance';
  TxTPlant_Heating_circuit_sObjectName                                   :T_BA_StateText:='HTC';
  TxTPlant_Heating_circuit_sDescription                                   :T_BA_StateText:='Heating circuit';
  TxTPlant_Heating_sObjectName                                           :T_BA_StateText:='HTG';
  TxTPlant_Heating_sDescription                                           :T_BA_StateText:='Heating';
  TxTPlant_Back_feed_system_sObjectName                                  :T_BA_StateText:='BSF';
  TxTPlant_Back_feed_system_sDescription                                  :T_BA_StateText:='Back-feed system';
  TxTPlant_Buffer_sObjectName                                            :T_BA_StateText:='BUF';
  TxTPlant_Buffer_sDescription                                            :T_BA_StateText:='Buffer';
  TxTPlant_Heat_distribution_network_sObjectName                         :T_BA_StateText:='HDN';
  TxTPlant_Heat_distribution_network_sDescription                         :T_BA_StateText:='Heat distribution network';
  TxTPlant_Heat_exchanger_sObjectName                                    :T_BA_StateText:='HEX';
  TxTPlant_Heat_exchanger_sDescription                                    :T_BA_StateText:='Heat exchanger';
// 423 Space-heating surfaces
  TxTPlant_Concrete_core_activation_sObjectName                          :T_BA_StateText:='CCA';
  TxTPlant_Concrete_core_activation_sDescription                          :T_BA_StateText:='Concrete core activation';
  TxTPlant_Overhead_heating_sObjectName                                  :T_BA_StateText:='OHH';
  TxTPlant_Overhead_heating_sDescription                                  :T_BA_StateText:='Overhead heating';
  TxTPlant_Ceiling_radiator_panels_sObjectName                           :T_BA_StateText:='CRP';
  TxTPlant_Ceiling_radiator_panels_sDescription                           :T_BA_StateText:='Ceiling radiator panels';
  TxTPlant_Facade_heating_sObjectName                                    :T_BA_StateText:='FAH';
  TxTPlant_Facade_heating_sDescription                                    :T_BA_StateText:='Facade heating';
  TxTPlant_Panel_heating_sObjectName                                     :T_BA_StateText:='PAH';
  TxTPlant_Panel_heating_sDescription                                     :T_BA_StateText:='Panel heating';
  TxTPlant_Underfloor_heating_sObjectName                                :T_BA_StateText:='UFH';
  TxTPlant_Underfloor_heating_sDescription                                :T_BA_StateText:='Underfloor heating';
  TxTPlant_Heated_chilled_ceiling_sObjectName                            :T_BA_StateText:='HCC';
  TxTPlant_Heated_chilled_ceiling_sDescription                            :T_BA_StateText:='Heated/chilled ceiling';
  TxTPlant_Static_heating_sObjectName                                    :T_BA_StateText:='STH';
  TxTPlant_Static_heating_sDescription                                    :T_BA_StateText:='Static heating';
// 430 Ventilation systems
  TxTPlant_Extract_air_system_sObjectName                                :T_BA_StateText:='EXS';
  TxTPlant_Extract_air_system_sDescription                                :T_BA_StateText:='Extract air system';
  TxTPlant_Roof_air_heater_sObjectName                                   :T_BA_StateText:='RAH';
  TxTPlant_Roof_air_heater_sDescription                                   :T_BA_StateText:='Roof air heater';
  TxTPlant_Circulatory_system_sObjectName                                :T_BA_StateText:='CCS';
  TxTPlant_Circulatory_system_sDescription                                :T_BA_StateText:='Circulatory system';
  TxTPlant_Air_processing_unit_sObjectName                               :T_BA_StateText:='APU';
  TxTPlant_Air_processing_unit_sDescription                               :T_BA_StateText:='Air processing unit';
  TxTPlant_Mechanical_smoke_extraction_system_sObjectName                :T_BA_StateText:='MSE';
  TxTPlant_Mechanical_smoke_extraction_system_sDescription                :T_BA_StateText:='Mechanical smoke extraction system';
  TxTPlant_Smoke_pressure_system_sObjectName                             :T_BA_StateText:='SPS';
  TxTPlant_Smoke_pressure_system_sDescription                             :T_BA_StateText:='Smoke pressure system';
  TxTPlant_Air_handling_unit_sObjectName                                 :T_BA_StateText:='AHU';
  TxTPlant_Air_handling_unit_sDescription                                 :T_BA_StateText:='Air handling unit';
  TxTPlant_Partial_air_conditioning_system_sObjectName                   :T_BA_StateText:='PAC';
  TxTPlant_Partial_air_conditioning_system_sDescription                   :T_BA_StateText:='Partial air-conditioning system';
  TxTPlant_Air_curtain_system_sObjectName                                :T_BA_StateText:='ACS';
  TxTPlant_Air_curtain_system_sDescription                                :T_BA_StateText:='Air curtain system';
  TxTPlant_Recirculating_air_system_sObjectName                          :T_BA_StateText:='RCA';
  TxTPlant_Recirculating_air_system_sDescription                          :T_BA_StateText:='Recirculating air system';
  TxTPlant_Full_air_conditioning_system_sObjectName                      :T_BA_StateText:='FAC';
  TxTPlant_Full_air_conditioning_system_sDescription                      :T_BA_StateText:='Full air-conditioning system';
  TxTPlant_Heat_recovery_system_sObjectName                              :T_BA_StateText:='REC';
  TxTPlant_Heat_recovery_system_sDescription                              :T_BA_StateText:='Heat recovery system';
  TxTPlant_Intake_air_system_sObjectName                                 :T_BA_StateText:='IAS';
  TxTPlant_Intake_air_system_sDescription                                 :T_BA_StateText:='Intake air system';
  TxTPlant_Smoke_extraction_system_sObjectName                           :T_BA_StateText:='SME';
  TxTPlant_Smoke_extraction_system_sDescription                           :T_BA_StateText:='Smoke extraction system';
// 434 Refrigeration systems
  TxTPlant_Remote_cooling_transfer_sObjectName                           :T_BA_StateText:='RCT';
  TxTPlant_Remote_cooling_transfer_sDescription                           :T_BA_StateText:='Remote cooling transfer';
  TxTPlant_Cooling_sObjectName                                           :T_BA_StateText:='COL';
  TxTPlant_Cooling_sDescription                                           :T_BA_StateText:='Cooling';
  TxTPlant_Cooling_circuit_sObjectName                                   :T_BA_StateText:='CCC';
  TxTPlant_Cooling_circuit_sDescription                                   :T_BA_StateText:='Cooling circuit';
  TxTPlant_Cooling_distribution_network_sObjectName                      :T_BA_StateText:='CDN';
  TxTPlant_Cooling_distribution_network_sDescription                      :T_BA_StateText:='Cooling distribution network';
  TxTPlant_Cold_water_generation_sObjectName                             :T_BA_StateText:='CWG';
  TxTPlant_Cold_water_generation_sDescription                             :T_BA_StateText:='Cold water generation';
  TxTPlant_Electrical_cabinet_cooling_sObjectName                        :T_BA_StateText:='ECC';
  TxTPlant_Electrical_cabinet_cooling_sDescription                        :T_BA_StateText:='Electrical cabinet cooling';
  TxTPlant_Cooling_storage_sObjectName                                   :T_BA_StateText:='CST';
  TxTPlant_Cooling_storage_sDescription                                   :T_BA_StateText:='Cooling storage';
  TxTPlant_Chilled_ceiling_sObjectName                                   :T_BA_StateText:='CHC';
  TxTPlant_Chilled_ceiling_sDescription                                   :T_BA_StateText:='Chilled ceiling';
  TxTPlant_Re_cooling_plant_sObjectName                                  :T_BA_StateText:='RCP';
  TxTPlant_Re_cooling_plant_sDescription                                  :T_BA_StateText:='Re-cooling plant';
// 441 High and medium-voltage systems
  TxTPlant_Switchgear_sObjectName                                        :T_BA_StateText:='SWG';
  TxTPlant_Switchgear_sDescription                                        :T_BA_StateText:='Switchgear';
  TxTPlant_Transformer_sObjectName                                       :T_BA_StateText:='TRF';
  TxTPlant_Transformer_sDescription                                       :T_BA_StateText:='Transformer';
  TxTPlant_Medium_voltage_system_sObjectName                             :T_BA_StateText:='MVS';
  TxTPlant_Medium_voltage_system_sDescription                             :T_BA_StateText:='Medium-voltage system';
  TxTPlant_Compensation_system_sObjectName                               :T_BA_StateText:='COS';
  TxTPlant_Compensation_system_sDescription                               :T_BA_StateText:='Compensation system';
  TxTPlant_Frequency_converter_system_sObjectName                        :T_BA_StateText:='FCS';
  TxTPlant_Frequency_converter_system_sDescription                        :T_BA_StateText:='Frequency converter system';
// 442 Self-power supply systems
  TxTPlant_Emissions_system_sObjectName                                  :T_BA_StateText:='EMS';
  TxTPlant_Emissions_system_sDescription                                  :T_BA_StateText:='Emissions system';
  TxTPlant_Battery_unit_sObjectName                                      :T_BA_StateText:='BAT';
  TxTPlant_Battery_unit_sDescription                                      :T_BA_StateText:='Battery unit';
  TxTPlant_Co_generation_unit_sObjectName                                :T_BA_StateText:='CGU';
  TxTPlant_Co_generation_unit_sDescription                                :T_BA_StateText:='Co-generation unit';
  TxTPlant_Fuel_supply_sObjectName                                       :T_BA_StateText:='FUS';
  TxTPlant_Fuel_supply_sDescription                                       :T_BA_StateText:='Fuel supply';
  TxTPlant_Standby_power_system_sObjectName                              :T_BA_StateText:='SPS';
  TxTPlant_Standby_power_system_sDescription                              :T_BA_StateText:='Standby power system';
  TxTPlant_Photovoltaic_system_sObjectName                               :T_BA_StateText:='PVS';
  TxTPlant_Photovoltaic_system_sDescription                               :T_BA_StateText:='Photovoltaic system';
  TxTPlant_Uninterruptible_power_supply_sObjectName                      :T_BA_StateText:='UPS';
  TxTPlant_Uninterruptible_power_supply_sDescription                      :T_BA_StateText:='Uninterruptible power supply';
// 443 Low-voltage switchgears
  TxTPlant_General_power_supply_sObjectName                              :T_BA_StateText:='GPS';
  TxTPlant_General_power_supply_sDescription                              :T_BA_StateText:='General power supply';
  TxTPlant_Safety_power_supply_sObjectName                               :T_BA_StateText:='SPO';
  TxTPlant_Safety_power_supply_sDescription                               :T_BA_StateText:='Safety power supply';
  TxTPlant_Lighting_sObjectName                                          :T_BA_StateText:='LIT';
  TxTPlant_Lighting_sDescription                                          :T_BA_StateText:='Lighting';
  TxTPlant_Emergency_lighting_sObjectName                                :T_BA_StateText:='EML';
  TxTPlant_Emergency_lighting_sDescription                                :T_BA_StateText:='Emergency lighting';
// 451 Telecommunications systems
  TxTPlant_Telecommunications_system_sObjectName                         :T_BA_StateText:='TEL';
  TxTPlant_Telecommunications_system_sDescription                         :T_BA_StateText:='Telecommunications system';
// 452 Search and signalling systems
  TxTPlant_Call_signalling_system_sObjectName                            :T_BA_StateText:='CSS';
  TxTPlant_Call_signalling_system_sDescription                            :T_BA_StateText:='Call signalling system';
  TxTPlant_Door_intercom_and_door_opener_system_sObjectName              :T_BA_StateText:='DIO';
  TxTPlant_Door_intercom_and_door_opener_system_sDescription              :T_BA_StateText:='Door intercom and door opener system';
  TxTPlant_Paging_system_sObjectName                                     :T_BA_StateText:='PGS';
  TxTPlant_Paging_system_sDescription                                     :T_BA_StateText:='Paging system';
// 453 Time service systems
  TxTPlant_Clock_and_time_recording_system_sObjectName                   :T_BA_StateText:='CTR';
  TxTPlant_Clock_and_time_recording_system_sDescription                   :T_BA_StateText:='Clock and time recording system';
// 454 Electro-acoustic systems
  TxTPlant_Electro_acoustic_sound_systems_sObjectName                    :T_BA_StateText:='ELA';
  TxTPlant_Electro_acoustic_sound_systems_sDescription                    :T_BA_StateText:='Electro-acoustic system, sound systems';
  TxTPlant_Conference_and_interpreting_equipment_sObjectName             :T_BA_StateText:='CIE';
  TxTPlant_Conference_and_interpreting_equipment_sDescription             :T_BA_StateText:='Conference and interpreting equipment';
  TxTPlant_Intercom_system_sObjectName                                   :T_BA_StateText:='ICS';
  TxTPlant_Intercom_system_sDescription                                   :T_BA_StateText:='Intercom system';
  TxTPlant_Voice_alarm_system_sObjectName                                :T_BA_StateText:='VAS';
  TxTPlant_Voice_alarm_system_sDescription                                :T_BA_StateText:='Voice alarm system';
  TxTPlant_Intercommunication_systems_sObjectName                        :T_BA_StateText:='ICS';
  TxTPlant_Intercommunication_systems_sDescription                        :T_BA_StateText:='Intercommunication systems';
// 455 Television and antenna systems
  TxTPlant_Television_system_sObjectName                                 :T_BA_StateText:='TVS';
  TxTPlant_Television_system_sDescription                                 :T_BA_StateText:='Television system';
  TxTPlant_Transmitting_and_receiving_antenna_system_sObjectName         :T_BA_StateText:='TRA';
  TxTPlant_Transmitting_and_receiving_antenna_system_sDescription         :T_BA_StateText:='Transmit. and receiving antenna system';
  TxTPlant_BOS_radio_system_sObjectName                                  :T_BA_StateText:='BOS';
  TxTPlant_BOS_radio_system_sDescription                                  :T_BA_StateText:='BOS radio system';
// 456 Hazard detection and alarm systems
  TxTPlant_Fire_detection_and_alarm_system_sObjectName                   :T_BA_StateText:='FDA';
  TxTPlant_Fire_detection_and_alarm_system_sDescription                   :T_BA_StateText:='Fire detection and alarm system';
  TxTPlant_Carbon_monoxide_warning_system_sObjectName                    :T_BA_StateText:='CMW';
  TxTPlant_Carbon_monoxide_warning_system_sDescription                    :T_BA_StateText:='Carbon monoxide warning system';
  TxTPlant_Burglar_alarm_system_sObjectName                              :T_BA_StateText:='BAS';
  TxTPlant_Burglar_alarm_system_sDescription                              :T_BA_StateText:='Burglar alarm system';
  TxTPlant_Fire_control_panel_sObjectName                                :T_BA_StateText:='FCP';
  TxTPlant_Fire_control_panel_sDescription                                :T_BA_StateText:='Fire control panel';
  TxTPlant_Escape_route_protection_system_sObjectName                    :T_BA_StateText:='ERP';
  TxTPlant_Escape_route_protection_system_sDescription                    :T_BA_StateText:='Escape route protection system';
  TxTPlant_Hazard_detection_system_sObjectName                           :T_BA_StateText:='HDS';
  TxTPlant_Hazard_detection_system_sDescription                           :T_BA_StateText:='Hazard detection system';
  TxTPlant_Gas_warning_system_sObjectName                                :T_BA_StateText:='GWS';
  TxTPlant_Gas_warning_system_sDescription                                :T_BA_StateText:='Gas warning system';
  TxTPlant_Smoke_aspiration_system_sObjectName                           :T_BA_StateText:='SAS';
  TxTPlant_Smoke_aspiration_system_sDescription                           :T_BA_StateText:='Smoke aspiration system';
  TxTPlant_Room_observation_system_sObjectName                           :T_BA_StateText:='ROS';
  TxTPlant_Room_observation_system_sDescription                           :T_BA_StateText:='Room observation system';
  TxTPlant_Robbery_alarm_system_sObjectName                              :T_BA_StateText:='ROA';
  TxTPlant_Robbery_alarm_system_sDescription                              :T_BA_StateText:='Robbery alarm system';
  TxTPlant_Guard_control_system_sObjectName                              :T_BA_StateText:='GCS';
  TxTPlant_Guard_control_system_sDescription                              :T_BA_StateText:='Guard control system';
  TxTPlant_Emergency_call_system_sObjectName                             :T_BA_StateText:='EMG';
  TxTPlant_Emergency_call_system_sDescription                             :T_BA_StateText:='Emergency call system';
  TxTPlant_Access_control_system_sObjectName                             :T_BA_StateText:='ACS';
  TxTPlant_Access_control_system_sDescription                             :T_BA_StateText:='Access control system';
// 457 Transmission grids
  TxTPlant_Networks_for_the_transmission_voice_text_etc_sObjectName      :T_BA_StateText:='LAN';
  TxTPlant_Networks_for_the_transmission_voice_text_etc_sDescription      :T_BA_StateText:='Networks  data, voice, text etc';
// 459 Telecommunication and information technology equipment, other
  TxTPlant_Remote_control_systems_sObjectName                            :T_BA_StateText:='RCS';
  TxTPlant_Remote_control_systems_sDescription                            :T_BA_StateText:='Remote control systems';
  TxTPlant_Parking_guidance_systems_sObjectName                          :T_BA_StateText:='PGS';
  TxTPlant_Parking_guidance_systems_sDescription                          :T_BA_StateText:='Parking guidance systems';
// 460 Conveyors
  TxTPlant_File_transportation_systems_sObjectName                       :T_BA_StateText:='FTS';
  TxTPlant_File_transportation_systems_sDescription                       :T_BA_StateText:='File transportation systems';
  TxTPlant_Lift_sObjectName                                              :T_BA_StateText:='LIF';
  TxTPlant_Lift_sDescription                                              :T_BA_StateText:='Lift';
  TxTPlant_Inspection_systems_sObjectName                                :T_BA_StateText:='ISS';
  TxTPlant_Inspection_systems_sDescription                                :T_BA_StateText:='Inspection systems';
  TxTPlant_Moving_walkways_sObjectName                                   :T_BA_StateText:='MWW';
  TxTPlant_Moving_walkways_sDescription                                   :T_BA_StateText:='Moving walkways';
  TxTPlant_Escalators_sObjectName                                        :T_BA_StateText:='ESC';
  TxTPlant_Escalators_sDescription                                        :T_BA_StateText:='Escalators';
  TxTPlant_External_lifts_sObjectName                                    :T_BA_StateText:='EXL';
  TxTPlant_External_lifts_sDescription                                    :T_BA_StateText:='External lifts';
  TxTPlant_Baggage_conveyor_system_sObjectName                           :T_BA_StateText:='BCS';
  TxTPlant_Baggage_conveyor_system_sDescription                           :T_BA_StateText:='Baggage conveyor system';
  TxTPlant_Pneumatic_delivery_systems_sObjectName                        :T_BA_StateText:='PDS';
  TxTPlant_Pneumatic_delivery_systems_sDescription                        :T_BA_StateText:='Pneumatic delivery systems';
  TxTPlant_Goods_transportation_facilities_sObjectName                   :T_BA_StateText:='GTF';
  TxTPlant_Goods_transportation_facilities_sDescription                   :T_BA_StateText:='Goods transportation facilities';
// 470 User-specific systems
// 471 Kitchen technology systems
  TxTPlant_Small_refrigeration_unit_sObjectName                          :T_BA_StateText:='SRU';
  TxTPlant_Small_refrigeration_unit_sDescription                          :T_BA_StateText:='Small refrigeration unit';
// 472 Laundry and cleaning systems
  TxTPlant_Disinfection_unit_sObjectName                                 :T_BA_StateText:='DIS';
  TxTPlant_Disinfection_unit_sDescription                                 :T_BA_StateText:='Disinfection unit';
  TxTPlant_Cleaning_unit_sObjectName                                     :T_BA_StateText:='CLU';
  TxTPlant_Cleaning_unit_sDescription                                     :T_BA_StateText:='Cleaning unit';
  TxTPlant_Sterilisation_systems_sObjectName                             :T_BA_StateText:='STR';
  TxTPlant_Sterilisation_systems_sDescription                             :T_BA_StateText:='Sterilisation systems';
  TxTPlant_Water_treatment_system_sObjectName                            :T_BA_StateText:='WTS';
  TxTPlant_Water_treatment_system_sDescription                            :T_BA_StateText:='Water treatment system';
  TxTPlant_Laundry_system_sObjectName                                    :T_BA_StateText:='LAU';
  TxTPlant_Laundry_system_sDescription                                    :T_BA_StateText:='Laundry system';
// 473 Media supply systems
  TxTPlant_Compressed_air_supply_system_sObjectName                      :T_BA_StateText:='COA';
  TxTPlant_Compressed_air_supply_system_sDescription                      :T_BA_StateText:='Compressed air supply system';
  TxTPlant_Pressure_regulator_unit_sObjectName                           :T_BA_StateText:='PRU';
  TxTPlant_Pressure_regulator_unit_sDescription                           :T_BA_StateText:='Pressure regulator unit';
  TxTPlant_Media_supply_system_sObjectName                               :T_BA_StateText:='MSS';
  TxTPlant_Media_supply_system_sDescription                               :T_BA_StateText:='Media supply system';
  TxTPlant_Medical_and_technical_gases_sObjectName                       :T_BA_StateText:='MTG';
  TxTPlant_Medical_and_technical_gases_sDescription                       :T_BA_StateText:='Medical and technical gases';
  TxTPlant_Vacuum_unit_sObjectName                                       :T_BA_StateText:='VAC';
  TxTPlant_Vacuum_unit_sDescription                                       :T_BA_StateText:='Vacuum unit';
// 474 Medical and laboratory equipment
  TxTPlant_Medical_technical_plant_sObjectName                           :T_BA_StateText:='MED';
  TxTPlant_Medical_technical_plant_sDescription                           :T_BA_StateText:='Medical technical plant';
  TxTPlant_Medical_gas_supply_sObjectName                                :T_BA_StateText:='MGS';
  TxTPlant_Medical_gas_supply_sDescription                                :T_BA_StateText:='Medical gas supply';
  TxTPlant_Laboratory_equipment_sObjectName                              :T_BA_StateText:='LAB';
  TxTPlant_Laboratory_equipment_sDescription                              :T_BA_StateText:='Laboratory equipment (general)';
// 475 Fire extinguishers
  TxTPlant_Fire_extinguisher_sObjectName                                 :T_BA_StateText:='FEG';
  TxTPlant_Fire_extinguisher_sDescription                                 :T_BA_StateText:='Fire extinguisher';
  TxTPlant_Gas_extinguishing_system_sObjectName                          :T_BA_StateText:='GES';
  TxTPlant_Gas_extinguishing_system_sDescription                          :T_BA_StateText:='Gas extinguishing system';
  TxTPlant_Fire_extinguishing_system_sObjectName                         :T_BA_StateText:='FES';
  TxTPlant_Fire_extinguishing_system_sDescription                         :T_BA_StateText:='Fire extinguishing system (general)';
  TxTPlant_Mist_extinguishing_system_sObjectName                         :T_BA_StateText:='MES';
  TxTPlant_Mist_extinguishing_system_sDescription                         :T_BA_StateText:='Mist-extinguishing system';
  TxTPlant_NOX_system_sObjectName                                        :T_BA_StateText:='NOX';
  TxTPlant_NOX_system_sDescription                                        :T_BA_StateText:='NOX system';
  TxTPlant_Sprinkler_system_sObjectName                                  :T_BA_StateText:='SPR';
  TxTPlant_Sprinkler_system_sDescription                                  :T_BA_StateText:='Sprinkler system';
  TxTPlant_Wall_hydrant_system_sObjectName                               :T_BA_StateText:='WHS';
  TxTPlant_Wall_hydrant_system_sDescription                               :T_BA_StateText:='Wall hydrant system';
// 478 Disposal facilities
  TxTPlant_Waste_disposal_system_sObjectName                             :T_BA_StateText:='WDS';
  TxTPlant_Waste_disposal_system_sDescription                             :T_BA_StateText:='Waste disposal system';
  TxTPlant_Media_disposal_system_sObjectName                             :T_BA_StateText:='MDS';
  TxTPlant_Media_disposal_system_sDescription                             :T_BA_StateText:='Media disposal system';
  TxTPlant_Vacuum_cleaning_systems_sObjectName                           :T_BA_StateText:='VCS';
  TxTPlant_Vacuum_cleaning_systems_sDescription                           :T_BA_StateText:='Vacuum cleaning systems';
// 480 Building automation and control systems
  TxTPlant_Information_focal_point_sObjectName                           :T_BA_StateText:='ISP';
  TxTPlant_Information_focal_point_sDescription                           :T_BA_StateText:='Information focal point';
  TxTPlant_Weather_station_sObjectName                                   :T_BA_StateText:='WET';
  TxTPlant_Weather_station_sDescription                                   :T_BA_StateText:='Weather station';
  TxTPlant_Management_and_operating_equipment_sObjectName                :T_BA_StateText:='MOE';
  TxTPlant_Management_and_operating_equipment_sDescription                :T_BA_StateText:='Management and operating equipment';
  TxTPlant_Room_automation_sObjectName                                   :T_BA_StateText:='RAU';
  TxTPlant_Room_automation_sDescription                                   :T_BA_StateText:='Room automation';
  TxTPlant_Room_automation_system_distributor_sObjectName                :T_BA_StateText:='RAS';
  TxTPlant_Room_automation_system_distributor_sDescription                :T_BA_StateText:='Room automation system distributor';
  TxTPlant_Control_cabinet_sObjectName                                   :T_BA_StateText:='CCB';
  TxTPlant_Control_cabinet_sDescription                                   :T_BA_StateText:='Control cabinet';
  TxTPlant_Settings_sObjectName                                          :T_BA_StateText:='SYP';
  TxTPlant_Settings_sDescription                                          :T_BA_StateText:='System parameters';
  TxTPlant_EventGroups_sObjectName                                       :T_BA_StateText:='EVG';
  TxTPlant_EventGroups_sDescription                                       :T_BA_StateText:='Event groups';
  TxTPlant_Global_Building_Data_sObjectName                              :T_BA_StateText:='GBD';
  TxTPlant_Global_Building_Data_sDescription                              :T_BA_StateText:='global building Data';
// 540 Technical equipment in outdoor facilities
  TxTPlant_Rainwater_retention_basin_sObjectName                         :T_BA_StateText:='RRB';
  TxTPlant_Rainwater_retention_basin_sDescription                         :T_BA_StateText:='Rainwater retention basin';
  TxTPlant_Cistern_system_sObjectName                                    :T_BA_StateText:='CIS';
  TxTPlant_Cistern_system_sDescription                                    :T_BA_StateText:='Cistern system';
END_VAR

// ---- Templates/GVLs/Language/English/TxtTrade_EN.TcGVL
{region '#Template'}
	{attribute 'Version' := '1.2.0.0'}
	{attribute 'Tags' := '"LCID": "1031", "Text": "GVL, DPAD, Trades, ObjectName, Description"'}
	{attribute 'Tags' := '"LCID": "1033", "Text": "GVL, DPAD, Trades, ObjectName, Description"'}
	{attribute 'Description' := '"LCID": "1031", "Text": "Textliste Gewerke"'}
	{attribute 'Description' := '"LCID": "1033", "Text": "Text list trades"'}
{endregion}

{attribute 'global_init_slot' := '40510'}
VAR_GLOBAL
  TxtTrade_Doors_gates_windows_sun_protection_sObjectName                :T_BA_StateText:='Doors, gates, windows, sun protection';
  TxtTrade_Doors_gates_windows_sun_protection_sDescription                :T_BA_StateText:='DGW';
  TxtTrade_Sewage_water_and_gas_plants_sObjectName                       :T_BA_StateText:='Sewage, water and gas plants';
  TxtTrade_Sewage_water_and_gas_plants_sDescription                       :T_BA_StateText:='SWG';
  TxtTrade_Heat_supply_systems_sObjectName                               :T_BA_StateText:='Heat supply systems';
  TxtTrade_Heat_supply_systems_sDescription                               :T_BA_StateText:='HTG';
  TxtTrade_Air_conditioning_sObjectName                                  :T_BA_StateText:='Air conditioning';
  TxtTrade_Air_conditioning_sDescription                                  :T_BA_StateText:='AC_';
  TxtTrade_Refrigeration_systems_sObjectName                             :T_BA_StateText:='Refrigeration systems';
  TxtTrade_Refrigeration_systems_sDescription                             :T_BA_StateText:='RFG';
  TxtTrade_High_voltage_systems_sObjectName                              :T_BA_StateText:='High-voltage systems';
  TxtTrade_High_voltage_systems_sDescription                              :T_BA_StateText:='HVS';
  TxtTrade_Telecommunication_and_information_technology_sObjectName      :T_BA_StateText:='Telecom. and information tech. equipment';
  TxtTrade_Telecommunication_and_information_technology_sDescription      :T_BA_StateText:='TIT';
  TxtTrade_Hazard_detection_and_alarm_systems_sObjectName                :T_BA_StateText:='Hazard detection and alarm systems';
  TxtTrade_Hazard_detection_and_alarm_systems_sDescription                :T_BA_StateText:='HDA';
  TxtTrade_Conveyors_sObjectName                                         :T_BA_StateText:='Conveyors';
  TxtTrade_Conveyors_sDescription                                         :T_BA_StateText:='CVY';
  TxtTrade_Kitchen_technology_systems_sObjectName                        :T_BA_StateText:='Kitchen technology systems';
  TxtTrade_Kitchen_technology_systems_sDescription                        :T_BA_StateText:='KTS';
  TxtTrade_Laundry_and_cleaning_systems_sObjectName                      :T_BA_StateText:='Laundry and cleaning systems';
  TxtTrade_Laundry_and_cleaning_systems_sDescription                      :T_BA_StateText:='LCS';
  TxtTrade_Media_supply_systems_sObjectName                              :T_BA_StateText:='Media supply systems';
  TxtTrade_Media_supply_systems_sDescription                              :T_BA_StateText:='MSS';
  TxtTrade_Medical_and_laboratory_equipment_sObjectName                  :T_BA_StateText:='Medical and laboratory equipment';
  TxtTrade_Medical_and_laboratory_equipment_sDescription                  :T_BA_StateText:='MED';
  TxtTrade_Fire_extinguishing_systems_sObjectName                        :T_BA_StateText:='Fire extinguishing systems';
  TxtTrade_Fire_extinguishing_systems_sDescription                        :T_BA_StateText:='FES';
  TxtTrade_Bathing_facilities_sObjectName                                :T_BA_StateText:='Bathing facilities';
  TxtTrade_Bathing_facilities_sDescription                                :T_BA_StateText:='BTF';
  TxtTrade_Process_heating_cooling_and_air_systems_sObjectName           :T_BA_StateText:='Process heating, cooling and air systems';
  TxtTrade_Process_heating_cooling_and_air_systems_sDescription           :T_BA_StateText:='PRO';
  TxtTrade_Waste_disposal_facilities_sObjectName                         :T_BA_StateText:='Waste disposal facilities';
  TxtTrade_Waste_disposal_facilities_sDescription                         :T_BA_StateText:='WDF';
  TxtTrade_Building_automation_and_control_systems_general_sObjectName   :T_BA_StateText:='Building automation  general';
  TxtTrade_Building_automation_and_control_systems_general_sDescription   :T_BA_StateText:='BAG';
  TxtTrade_Automation_focal_point_information_focal_point_sObjectName    :T_BA_StateText:='Automation focal point';
  TxtTrade_Automation_focal_point_information_focal_point_sDescription    :T_BA_StateText:='AFP';
  TxtTrade_Room_automation_sObjectName                                   :T_BA_StateText:='Room automation';
  TxtTrade_Room_automation_sDescription                                   :T_BA_StateText:='ROM';
  TxtTrade_Outdoor_devices_sObjectName                                   :T_BA_StateText:='Outdoor devices';
  TxtTrade_Outdoor_devices_sDescription                                   :T_BA_StateText:='ODD';
END_VAR

// ---- Templates/GVLs/Language/German/LblAggregates_DE.TcGVL
{region '#Template'}
	{attribute 'Version' := '1.2.0.0'}
	{attribute 'Tags' := '"LCID": "1031", "Text": "GVL, AKS, Labels, ObjectName, Description"'}
	{attribute 'Tags' := '"LCID": "1033", "Text": "GVL, DPAD, Labels, ObjectName, Description"'}
	{attribute 'Description' := '"LCID": "1031", "Text": "Anlagenkennzeichnungssystem, Labels Aggregate"'}
	{attribute 'Description' := '"LCID": "1033", "Text": "Data Point Addressing Description, Labels aggregate"'}
{endregion}

